SUBAPPLICATION Uebung_000 (* ADD *)
  (* Standard: 61499-2; Description: Copyright (c) 2023 Meisterschulen am Ostbahnhof This program and the accompanying materials are made available under the terms of the Eclipse Public License 2.0 which is available at https://www.eclipse.org/legal/epl-2.0/ SPDX-License-Identifier: EPL-2.0 *)
  (* Version 1.0, 2023-10-23, Franz Höpfinger, Meisterschulen am Ostbahnhof *)
  PACKAGE Uebungen;
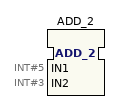
  FBS
    ADD_2 : iec61131::arithmetic::ADD_2(IN1 := INT#5, IN2 := INT#3);
  END_FBS
END_SUBAPPLICATION
